TYPE Item :
STRUCT
END_STRUCT
END_TYPE

(* stored: Version 1.1.0.1, ProductVersion 3.1.4024.13
   DUT Item: Id {d87c8f71-ff87-4174-a5f9-0bd3b17618c6} *)
